KUKA KRL program: ps_l_res_c1.src, ps_l_res_c1.dat

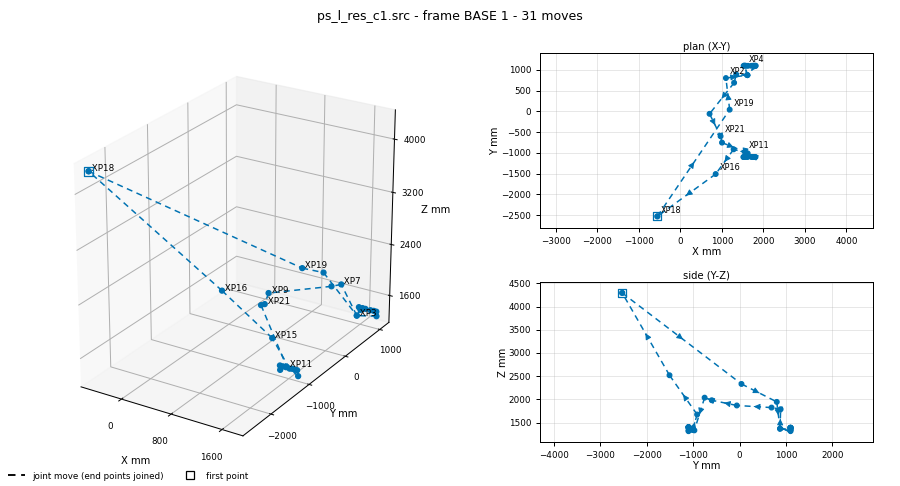
[picture p0: tool path of ps_l_res_c1.src in frame BASE 1, 31 of 31 moves have a stored position in this frame; points joined in program order, loops and branches not executed]
--- ps_l_res_c1.src ---
&ACCESS RVO1
&REL 7
&COMMENT SOLDA GUN C1 SEM GRIPPER
&PARAM DISKPATH = KRC:\R1\Program
DEF ps_l_res_c1( )
;FOLD INI
;FOLD SPOTTECH INI
USERSPOT(#INIT)
;ENDFOLD (SPOTTECH INI)
;FOLD GRIPPERTECH INI
USER_GRP(0,DUMMY,DUMMY,GDEFAULT)
;ENDFOLD (GRIPPERTECH INI)
  ;FOLD USER INI
    ;Make your modifications here

  ;ENDFOLD (USER INI)
;ENDFOLD (INI)

; Caracterização dos meios de produção:
; Versão Atual:
; 15/07/2013 12:00 Name: P13.050-R5 CHANGES: Solda Respot Actros
; C1 LTA/LTB/MGS/MGSB

chk_w1_wechs_ok ( )      ; CHECK FERRAMENTA: C1

;FOLD PTP P18 CONT Vel=100 % PDAT31 Tool[1]:Gun C1 Base[1]:ACTROS;%{PE}%R 8.2.20,%MKUKATPBASIS,%CMOVE,%VPTP,%P 1:PTP, 2:P18, 3:C_DIS, 5:100, 7:PDAT31
$BWDSTART=FALSE
PDAT_ACT=PPDAT31
FDAT_ACT=FP18
BAS(#PTP_PARAMS,100)
PTP XP18 C_DIS
;ENDFOLD

if MaxStandMenge (1) then
 MaxStandmengeErreicht (1)
endif

IF (NOT(GHOST())) THEN
if Elektrodenwechsel (1) then
 e_fraes1 ()
endif
ENDIF

;FOLD PTP P19 CONT Vel=100 % PDAT32 Tool[1]:Gun C1 Base[1]:ACTROS;%{PE}%R 8.2.20,%MKUKATPBASIS,%CMOVE,%VPTP,%P 1:PTP, 2:P19, 3:C_DIS, 5:100, 7:PDAT32
$BWDSTART=FALSE
PDAT_ACT=PPDAT32
FDAT_ACT=FP19
BAS(#PTP_PARAMS,100)
PTP XP19 C_DIS
;ENDFOLD

;FOLD OUT 3334 'R5 solicita lib soldar respot' State=TRUE ;%{PE}%R 8.2.20,%MKUKATPBASIS,%COUT,%VOUTX,%P 2:3334, 3:R5 solicita lib soldar respot, 5:TRUE, 6:
$OUT[3334]=TRUE
;ENDFOLD
;FOLD OUT 3337 'R5 retirando garra Geo' State=TRUE ;%{PE}%R 8.2.20,%MKUKATPBASIS,%COUT,%VOUTX,%P 2:3337, 3:R5 retirando garra Geo, 5:TRUE, 6:
$OUT[3337]=TRUE
;ENDFOLD
;FOLD WAIT FOR ( IN 3334 'Aguarda lib soldar respot' );%{PE}%R 8.2.20,%MKUKATPBASIS,%CEXT_WAIT_FOR,%VEXT_WAIT_FOR,%P 2:, 4:, 5:$IN, 6:3334, 7:Aguarda lib soldar respot, 9:
WAIT FOR  ( $IN[3334] )
;ENDFOLD
;FOLD OUT 3334 'R5 solicita lib soldar respot' State=FALSE ;%{PE}%R 8.2.20,%MKUKATPBASIS,%COUT,%VOUTX,%P 2:3334, 3:R5 solicita lib soldar respot, 5:FALSE, 6:
$OUT[3334]=FALSE
;ENDFOLD
;FOLD OUT 3337 'R5 retirando garra Geo' State=FALSE ;%{PE}%R 8.2.20,%MKUKATPBASIS,%COUT,%VOUTX,%P 2:3337, 3:R5 retirando garra Geo, 5:FALSE, 6:
$OUT[3337]=FALSE
;ENDFOLD
;FOLD OUT 3338 'R5 solda geometria concluida' State=FALSE ;%{PE}%R 8.2.20,%MKUKATPBASIS,%COUT,%VOUTX,%P 2:3338, 3:R5 solda geometria concluida, 5:FALSE, 6:
$OUT[3338]=FALSE
;ENDFOLD
;FOLD OUT 3348 'Fora area GEOBOX' State=FALSE ;%{PE}%R 8.2.20,%MKUKATPBASIS,%COUT,%VOUTX,%P 2:3348, 3:Fora area GEOBOX, 5:FALSE, 6:
$OUT[3348]=FALSE
;ENDFOLD
;FOLD  ;%{PE}%R 8.2.20,%MKUKATPBASIS,%CCOMMENT,%VNORMAL,%P 2:
;ENDFOLD
;FOLD PTP P2 CONT Vel=100 % PDAT2 Tool[1]:Gun C1 Base[1]:ACTROS;%{PE}%R 8.2.20,%MKUKATPBASIS,%CMOVE,%VPTP,%P 1:PTP, 2:P2, 3:C_DIS, 5:100, 7:PDAT2
$BWDSTART=FALSE
PDAT_ACT=PPDAT2
FDAT_ACT=FP2
BAS(#PTP_PARAMS,100)
PTP XP2 C_DIS
;ENDFOLD
;FOLD PTP P3 CONT Vel=100 % PDAT3 Tool[1]:Gun C1 Base[1]:ACTROS;%{PE}%R 8.2.20,%MKUKATPBASIS,%CMOVE,%VPTP,%P 1:PTP, 2:P3, 3:C_DIS, 5:100, 7:PDAT3
$BWDSTART=FALSE
PDAT_ACT=PPDAT3
FDAT_ACT=FP3
BAS(#PTP_PARAMS,100)
PTP XP3 C_DIS
;ENDFOLD
;FOLD PTP P4 CONT Vel=100 % PDAT4 Tool[1]:Gun C1 Base[1]:ACTROS;%{PE}%R 8.2.20,%MKUKATPBASIS,%CMOVE,%VPTP,%P 1:PTP, 2:P4, 3:C_DIS, 5:100, 7:PDAT4
$BWDSTART=FALSE
PDAT_ACT=PPDAT4
FDAT_ACT=FP4
BAS(#PTP_PARAMS,100)
PTP XP4 C_DIS
;ENDFOLD

;FOLD ; swp_60_5662;%{PE}%R 8.2.20,%MKUKATPBASIS,%CCOMMENT,%VNORMAL,%P 2:swp_60_5662
;ENDFOLD
;FOLD PTP Xswp_60_5662 PDAT5 SPOT Gun=1 RETR OPN PgNo1=38 ACTIVE=1 Tool[1]:Gun C1 Base[1]:ACTROS;%{PE}%R 8.2.2,%MKUKATPSPOT,%CSPOT,%VPTP,%P 1:PTP, 2:Xswp_60_5662, 3:, 5:100, 7:PDAT5, 10:1, 12:#FIRST, 14:#OPN, 16:38, 18:1, 20:0, 22:0, 24:1, 25:NORMAL
$BWDSTART=FALSE
PDAT_ACT=PPDAT5
FDAT_ACT=FXswp_60_5662
BAS(#PTP_PARAMS,PPDAT5.VEL)
S_ACT.GUN=1
S_ACT.PAIR=SDEFAULT.PAIR
S_ACT.RETR=#OPN
S_ACT.CLO_TM=1
S_ACT.PGNO1=38
S_ACT.PGNO2=SDEFAULT.PGNO2
S_ACT.PRESS1=SDEFAULT.PRESS1
S_ACT.PRESS2=SDEFAULT.PRESS2
S_READY=FALSE
PTP XXswp_60_5662
USERSPOT(#SPOT, S_ACT)
WAIT FOR S_READY
;ENDFOLD

;FOLD ; swp_60_5664;%{PE}%R 8.2.20,%MKUKATPBASIS,%CCOMMENT,%VNORMAL,%P 2:swp_60_5664
;ENDFOLD
;FOLD PTP Xswp_60_5664 PDAT7 SPOT Gun=1 RETR CLS PgNo1=39 ACTIVE=1 Tool[1]:Gun C1 Base[1]:ACTROS;%{PE}%R 8.2.2,%MKUKATPSPOT,%CSPOT,%VPTP,%P 1:PTP, 2:Xswp_60_5664, 3:, 5:100, 7:PDAT7, 10:1, 12:#FIRST, 14:#CLO, 16:39, 18:1, 20:0, 22:0, 24:1, 25:NORMAL
$BWDSTART=FALSE
PDAT_ACT=PPDAT7
FDAT_ACT=FXswp_60_5664
BAS(#PTP_PARAMS,PPDAT7.VEL)
S_ACT.GUN=1
S_ACT.PAIR=SDEFAULT.PAIR
S_ACT.RETR=#CLO
S_ACT.CLO_TM=1
S_ACT.PGNO1=39
S_ACT.PGNO2=SDEFAULT.PGNO2
S_ACT.PRESS1=SDEFAULT.PRESS1
S_ACT.PRESS2=SDEFAULT.PRESS2
S_READY=FALSE
PTP XXswp_60_5664
USERSPOT(#SPOT, S_ACT)
WAIT FOR S_READY
;ENDFOLD

;FOLD ; swp_60_5666;%{PE}%R 8.2.20,%MKUKATPBASIS,%CCOMMENT,%VNORMAL,%P 2:swp_60_5666
;ENDFOLD
;FOLD PTP Xswp_60_5666 PDAT6 SPOT Gun=1 RETR CLS PgNo1=40 ACTIVE=1 Tool[1]:Gun C1 Base[1]:ACTROS;%{PE}%R 8.2.2,%MKUKATPSPOT,%CSPOT,%VPTP,%P 1:PTP, 2:Xswp_60_5666, 3:, 5:100, 7:PDAT6, 10:1, 12:#FIRST, 14:#CLO, 16:40, 18:1, 20:0, 22:0, 24:1, 25:NORMAL
$BWDSTART=FALSE
PDAT_ACT=PPDAT6
FDAT_ACT=FXswp_60_5666
BAS(#PTP_PARAMS,PPDAT6.VEL)
S_ACT.GUN=1
S_ACT.PAIR=SDEFAULT.PAIR
S_ACT.RETR=#CLO
S_ACT.CLO_TM=1
S_ACT.PGNO1=40
S_ACT.PGNO2=SDEFAULT.PGNO2
S_ACT.PRESS1=SDEFAULT.PRESS1
S_ACT.PRESS2=SDEFAULT.PRESS2
S_READY=FALSE
PTP XXswp_60_5666
USERSPOT(#SPOT, S_ACT)
WAIT FOR S_READY
;ENDFOLD

;FOLD ; swp_60_5670;%{PE}%R 8.2.20,%MKUKATPBASIS,%CCOMMENT,%VNORMAL,%P 2:swp_60_5670
;ENDFOLD
;FOLD PTP Xswp_60_5670 PDAT8 SPOT Gun=1 RETR CLS PgNo1=41 ACTIVE=1 Tool[1]:Gun C1 Base[1]:ACTROS;%{PE}%R 8.2.2,%MKUKATPSPOT,%CSPOT,%VPTP,%P 1:PTP, 2:Xswp_60_5670, 3:, 5:100, 7:PDAT8, 10:1, 12:#FIRST, 14:#CLO, 16:41, 18:1, 20:0, 22:0, 24:1, 25:NORMAL
$BWDSTART=FALSE
PDAT_ACT=PPDAT8
FDAT_ACT=FXswp_60_5670
BAS(#PTP_PARAMS,PPDAT8.VEL)
S_ACT.GUN=1
S_ACT.PAIR=SDEFAULT.PAIR
S_ACT.RETR=#CLO
S_ACT.CLO_TM=1
S_ACT.PGNO1=41
S_ACT.PGNO2=SDEFAULT.PGNO2
S_ACT.PRESS1=SDEFAULT.PRESS1
S_ACT.PRESS2=SDEFAULT.PRESS2
S_READY=FALSE
PTP XXswp_60_5670
USERSPOT(#SPOT, S_ACT)
WAIT FOR S_READY
;ENDFOLD

;FOLD ; swp_60_5672;%{PE}%R 8.2.20,%MKUKATPBASIS,%CCOMMENT,%VNORMAL,%P 2:swp_60_5672
;ENDFOLD
;FOLD PTP SWP_60_5672 PDAT30 SPOT Gun=1 RETR CLS PgNo1=42 ACTIVE=1 Tool[1]:Gun C1 Base[1]:ACTROS;%{PE}%R 8.2.2,%MKUKATPSPOT,%CSPOT,%VPTP,%P 1:PTP, 2:SWP_60_5672, 3:, 5:100, 7:PDAT30, 10:1, 12:#FIRST, 14:#CLO, 16:42, 18:1, 20:0, 22:0, 24:1, 25:NORMAL
$BWDSTART=FALSE
PDAT_ACT=PPDAT30
FDAT_ACT=FSWP_60_5672
BAS(#PTP_PARAMS,PPDAT30.VEL)
S_ACT.GUN=1
S_ACT.PAIR=SDEFAULT.PAIR
S_ACT.RETR=#CLO
S_ACT.CLO_TM=1
S_ACT.PGNO1=42
S_ACT.PGNO2=SDEFAULT.PGNO2
S_ACT.PRESS1=SDEFAULT.PRESS1
S_ACT.PRESS2=SDEFAULT.PRESS2
S_READY=FALSE
PTP XSWP_60_5672
USERSPOT(#SPOT, S_ACT)
WAIT FOR S_READY
;ENDFOLD

;FOLD ; swp_60_5674;%{PE}%R 8.2.20,%MKUKATPBASIS,%CCOMMENT,%VNORMAL,%P 2:swp_60_5674
;ENDFOLD
;FOLD PTP Xswp_60_5674 PDAT10 SPOT Gun=1 RETR CLS PgNo1=43 ACTIVE=1 Tool[1]:Gun C1 Base[1]:ACTROS;%{PE}%R 8.2.2,%MKUKATPSPOT,%CSPOT,%VPTP,%P 1:PTP, 2:Xswp_60_5674, 3:, 5:100, 7:PDAT10, 10:1, 12:#FIRST, 14:#CLO, 16:43, 18:1, 20:0, 22:0, 24:1, 25:NORMAL
$BWDSTART=FALSE
PDAT_ACT=PPDAT10
FDAT_ACT=FXswp_60_5674
BAS(#PTP_PARAMS,PPDAT10.VEL)
S_ACT.GUN=1
S_ACT.PAIR=SDEFAULT.PAIR
S_ACT.RETR=#CLO
S_ACT.CLO_TM=1
S_ACT.PGNO1=43
S_ACT.PGNO2=SDEFAULT.PGNO2
S_ACT.PRESS1=SDEFAULT.PRESS1
S_ACT.PRESS2=SDEFAULT.PRESS2
S_READY=FALSE
PTP XXswp_60_5674
USERSPOT(#SPOT, S_ACT)
WAIT FOR S_READY
;ENDFOLD

;FOLD PTP P5 CONT Vel=100 % PDAT11 Tool[1]:Gun C1 Base[1]:ACTROS;%{PE}%R 8.2.20,%MKUKATPBASIS,%CMOVE,%VPTP,%P 1:PTP, 2:P5, 3:C_DIS, 5:100, 7:PDAT11
$BWDSTART=FALSE
PDAT_ACT=PPDAT11
FDAT_ACT=FP5
BAS(#PTP_PARAMS,100)
PTP XP5 C_DIS
;ENDFOLD
;FOLD PTP P6 CONT Vel=100 % PDAT12 Tool[1]:Gun C1 Base[1]:ACTROS;%{PE}%R 8.2.20,%MKUKATPBASIS,%CMOVE,%VPTP,%P 1:PTP, 2:P6, 3:C_DIS, 5:100, 7:PDAT12
$BWDSTART=FALSE
PDAT_ACT=PPDAT12
FDAT_ACT=FP6
BAS(#PTP_PARAMS,100)
PTP XP6 C_DIS
;ENDFOLD
;FOLD PTP P7 CONT Vel=100 % PDAT13 Tool[1]:Gun C1 Base[1]:ACTROS;%{PE}%R 8.2.20,%MKUKATPBASIS,%CMOVE,%VPTP,%P 1:PTP, 2:P7, 3:C_DIS, 5:100, 7:PDAT13
$BWDSTART=FALSE
PDAT_ACT=PPDAT13
FDAT_ACT=FP7
BAS(#PTP_PARAMS,100)
PTP XP7 C_DIS
;ENDFOLD
;FOLD PTP P22 CONT Vel=100 % PDAT35 Tool[1]:Gun C1 Base[1]:ACTROS;%{PE}%R 8.2.20,%MKUKATPBASIS,%CMOVE,%VPTP,%P 1:PTP, 2:P22, 3:C_DIS, 5:100, 7:PDAT35
$BWDSTART=FALSE
PDAT_ACT=PPDAT35
FDAT_ACT=FP22
BAS(#PTP_PARAMS,100)
PTP XP22 C_DIS
;ENDFOLD
;FOLD PTP P9 CONT Vel=100 % PDAT15 Tool[1]:Gun C1 Base[1]:ACTROS;%{PE}%R 8.2.20,%MKUKATPBASIS,%CMOVE,%VPTP,%P 1:PTP, 2:P9, 3:C_DIS, 5:100, 7:PDAT15
$BWDSTART=FALSE
PDAT_ACT=PPDAT15
FDAT_ACT=FP9
BAS(#PTP_PARAMS,100)
PTP XP9 C_DIS
;ENDFOLD
;FOLD PTP P21 CONT Vel=100 % PDAT34 Tool[1]:Gun C1 Base[1]:ACTROS;%{PE}%R 8.2.20,%MKUKATPBASIS,%CMOVE,%VPTP,%P 1:PTP, 2:P21, 3:C_DIS, 5:100, 7:PDAT34
$BWDSTART=FALSE
PDAT_ACT=PPDAT34
FDAT_ACT=FP21
BAS(#PTP_PARAMS,100)
PTP XP21 C_DIS
;ENDFOLD
;FOLD PTP P10 CONT Vel=100 % PDAT16 Tool[1]:Gun C1 Base[1]:ACTROS;%{PE}%R 8.2.20,%MKUKATPBASIS,%CMOVE,%VPTP,%P 1:PTP, 2:P10, 3:C_DIS, 5:100, 7:PDAT16
$BWDSTART=FALSE
PDAT_ACT=PPDAT16
FDAT_ACT=FP10
BAS(#PTP_PARAMS,100)
PTP XP10 C_DIS
;ENDFOLD
;FOLD PTP P11 CONT Vel=100 % PDAT17 Tool[1]:Gun C1 Base[1]:ACTROS;%{PE}%R 8.2.20,%MKUKATPBASIS,%CMOVE,%VPTP,%P 1:PTP, 2:P11, 3:C_DIS, 5:100, 7:PDAT17
$BWDSTART=FALSE
PDAT_ACT=PPDAT17
FDAT_ACT=FP11
BAS(#PTP_PARAMS,100)
PTP XP11 C_DIS
;ENDFOLD
;FOLD PTP P12 CONT Vel=100 % PDAT18 Tool[1]:Gun C1 Base[1]:ACTROS;%{PE}%R 8.2.20,%MKUKATPBASIS,%CMOVE,%VPTP,%P 1:PTP, 2:P12, 3:C_DIS, 5:100, 7:PDAT18
$BWDSTART=FALSE
PDAT_ACT=PPDAT18
FDAT_ACT=FP12
BAS(#PTP_PARAMS,100)
PTP XP12 C_DIS
;ENDFOLD

;FOLD ; swp_60_5661;%{PE}%R 8.2.20,%MKUKATPBASIS,%CCOMMENT,%VNORMAL,%P 2:swp_60_5661
;ENDFOLD
;FOLD PTP Xswp_60_5661 PDAT19 SPOT Gun=1 RETR CLS PgNo1=44 ACTIVE=1 Tool[1]:Gun C1 Base[1]:ACTROS;%{PE}%R 8.2.2,%MKUKATPSPOT,%CSPOT,%VPTP,%P 1:PTP, 2:Xswp_60_5661, 3:, 5:100, 7:PDAT19, 10:1, 12:#FIRST, 14:#CLO, 16:44, 18:1, 20:0, 22:0, 24:1, 25:NORMAL
$BWDSTART=FALSE
PDAT_ACT=PPDAT19
FDAT_ACT=FXswp_60_5661
BAS(#PTP_PARAMS,PPDAT19.VEL)
S_ACT.GUN=1
S_ACT.PAIR=SDEFAULT.PAIR
S_ACT.RETR=#CLO
S_ACT.CLO_TM=1
S_ACT.PGNO1=44
S_ACT.PGNO2=SDEFAULT.PGNO2
S_ACT.PRESS1=SDEFAULT.PRESS1
S_ACT.PRESS2=SDEFAULT.PRESS2
S_READY=FALSE
PTP XXswp_60_5661
USERSPOT(#SPOT, S_ACT)
WAIT FOR S_READY
;ENDFOLD

;FOLD ; swp_60_5663;%{PE}%R 8.2.20,%MKUKATPBASIS,%CCOMMENT,%VNORMAL,%P 2:swp_60_5663
;ENDFOLD
;FOLD PTP Xswp_60_5663 PDAT20 SPOT Gun=1 RETR CLS PgNo1=45 ACTIVE=1 Tool[1]:Gun C1 Base[1]:ACTROS;%{PE}%R 8.2.2,%MKUKATPSPOT,%CSPOT,%VPTP,%P 1:PTP, 2:Xswp_60_5663, 3:, 5:100, 7:PDAT20, 10:1, 12:#FIRST, 14:#CLO, 16:45, 18:1, 20:0, 22:0, 24:1, 25:NORMAL
$BWDSTART=FALSE
PDAT_ACT=PPDAT20
FDAT_ACT=FXswp_60_5663
BAS(#PTP_PARAMS,PPDAT20.VEL)
S_ACT.GUN=1
S_ACT.PAIR=SDEFAULT.PAIR
S_ACT.RETR=#CLO
S_ACT.CLO_TM=1
S_ACT.PGNO1=45
S_ACT.PGNO2=SDEFAULT.PGNO2
S_ACT.PRESS1=SDEFAULT.PRESS1
S_ACT.PRESS2=SDEFAULT.PRESS2
S_READY=FALSE
PTP XXswp_60_5663
USERSPOT(#SPOT, S_ACT)
WAIT FOR S_READY
;ENDFOLD

;FOLD ; swp_60_5665;%{PE}%R 8.2.20,%MKUKATPBASIS,%CCOMMENT,%VNORMAL,%P 2:swp_60_5665
;ENDFOLD
;FOLD PTP Xswp_60_5665 PDAT21 SPOT Gun=1 RETR CLS PgNo1=46 ACTIVE=1 Tool[1]:Gun C1 Base[1]:ACTROS;%{PE}%R 8.2.2,%MKUKATPSPOT,%CSPOT,%VPTP,%P 1:PTP, 2:Xswp_60_5665, 3:, 5:100, 7:PDAT21, 10:1, 12:#FIRST, 14:#CLO, 16:46, 18:1, 20:0, 22:0, 24:1, 25:NORMAL
$BWDSTART=FALSE
PDAT_ACT=PPDAT21
FDAT_ACT=FXswp_60_5665
BAS(#PTP_PARAMS,PPDAT21.VEL)
S_ACT.GUN=1
S_ACT.PAIR=SDEFAULT.PAIR
S_ACT.RETR=#CLO
S_ACT.CLO_TM=1
S_ACT.PGNO1=46
S_ACT.PGNO2=SDEFAULT.PGNO2
S_ACT.PRESS1=SDEFAULT.PRESS1
S_ACT.PRESS2=SDEFAULT.PRESS2
S_READY=FALSE
PTP XXswp_60_5665
USERSPOT(#SPOT, S_ACT)
WAIT FOR S_READY
;ENDFOLD

;FOLD ; swp_60_5669;%{PE}%R 8.2.20,%MKUKATPBASIS,%CCOMMENT,%VNORMAL,%P 2:swp_60_5669
;ENDFOLD
;FOLD PTP Xswp_60_5669 PDAT22 SPOT Gun=1 RETR CLS PgNo1=47 ACTIVE=1 Tool[1]:Gun C1 Base[1]:ACTROS;%{PE}%R 8.2.2,%MKUKATPSPOT,%CSPOT,%VPTP,%P 1:PTP, 2:Xswp_60_5669, 3:, 5:100, 7:PDAT22, 10:1, 12:#FIRST, 14:#CLO, 16:47, 18:1, 20:0, 22:0, 24:1, 25:NORMAL
$BWDSTART=FALSE
PDAT_ACT=PPDAT22
FDAT_ACT=FXswp_60_5669
BAS(#PTP_PARAMS,PPDAT22.VEL)
S_ACT.GUN=1
S_ACT.PAIR=SDEFAULT.PAIR
S_ACT.RETR=#CLO
S_ACT.CLO_TM=1
S_ACT.PGNO1=47
S_ACT.PGNO2=SDEFAULT.PGNO2
S_ACT.PRESS1=SDEFAULT.PRESS1
S_ACT.PRESS2=SDEFAULT.PRESS2
S_READY=FALSE
PTP XXswp_60_5669
USERSPOT(#SPOT, S_ACT)
WAIT FOR S_READY
;ENDFOLD

;FOLD ; swp_60_5671;%{PE}%R 8.2.20,%MKUKATPBASIS,%CCOMMENT,%VNORMAL,%P 2:swp_60_5671
;ENDFOLD
;FOLD PTP Xswp_60_5671 PDAT23 SPOT Gun=1 RETR CLS PgNo1=48 ACTIVE=1 Tool[1]:Gun C1 Base[1]:ACTROS;%{PE}%R 8.2.2,%MKUKATPSPOT,%CSPOT,%VPTP,%P 1:PTP, 2:Xswp_60_5671, 3:, 5:100, 7:PDAT23, 10:1, 12:#FIRST, 14:#CLO, 16:48, 18:1, 20:0, 22:0, 24:1, 25:NORMAL
$BWDSTART=FALSE
PDAT_ACT=PPDAT23
FDAT_ACT=FXswp_60_5671
BAS(#PTP_PARAMS,PPDAT23.VEL)
S_ACT.GUN=1
S_ACT.PAIR=SDEFAULT.PAIR
S_ACT.RETR=#CLO
S_ACT.CLO_TM=1
S_ACT.PGNO1=48
S_ACT.PGNO2=SDEFAULT.PGNO2
S_ACT.PRESS1=SDEFAULT.PRESS1
S_ACT.PRESS2=SDEFAULT.PRESS2
S_READY=FALSE
PTP XXswp_60_5671
USERSPOT(#SPOT, S_ACT)
WAIT FOR S_READY
;ENDFOLD

;FOLD ; swp_60_5673;%{PE}%R 8.2.20,%MKUKATPBASIS,%CCOMMENT,%VNORMAL,%P 2:swp_60_5673
;ENDFOLD
;FOLD PTP Xswp_60_5673 PDAT24 SPOT Gun=1 RETR OPN PgNo1=49 ACTIVE=1 Tool[1]:Gun C1 Base[1]:ACTROS;%{PE}%R 8.2.2,%MKUKATPSPOT,%CSPOT,%VPTP,%P 1:PTP, 2:Xswp_60_5673, 3:, 5:100, 7:PDAT24, 10:1, 12:#FIRST, 14:#OPN, 16:49, 18:1, 20:0, 22:0, 24:1, 25:NORMAL
$BWDSTART=FALSE
PDAT_ACT=PPDAT24
FDAT_ACT=FXswp_60_5673
BAS(#PTP_PARAMS,PPDAT24.VEL)
S_ACT.GUN=1
S_ACT.PAIR=SDEFAULT.PAIR
S_ACT.RETR=#OPN
S_ACT.CLO_TM=1
S_ACT.PGNO1=49
S_ACT.PGNO2=SDEFAULT.PGNO2
S_ACT.PRESS1=SDEFAULT.PRESS1
S_ACT.PRESS2=SDEFAULT.PRESS2
S_READY=FALSE
PTP XXswp_60_5673
USERSPOT(#SPOT, S_ACT)
WAIT FOR S_READY
;ENDFOLD

;FOLD PTP P13 CONT Vel=100 % PDAT25 Tool[1]:Gun C1 Base[1]:ACTROS;%{PE}%R 8.2.20,%MKUKATPBASIS,%CMOVE,%VPTP,%P 1:PTP, 2:P13, 3:C_DIS, 5:100, 7:PDAT25
$BWDSTART=FALSE
PDAT_ACT=PPDAT25
FDAT_ACT=FP13
BAS(#PTP_PARAMS,100)
PTP XP13 C_DIS
;ENDFOLD
;FOLD PTP P14 CONT Vel=100 % PDAT26 Tool[1]:Gun C1 Base[1]:ACTROS;%{PE}%R 8.2.20,%MKUKATPBASIS,%CMOVE,%VPTP,%P 1:PTP, 2:P14, 3:C_DIS, 5:100, 7:PDAT26
$BWDSTART=FALSE
PDAT_ACT=PPDAT26
FDAT_ACT=FP14
BAS(#PTP_PARAMS,100)
PTP XP14 C_DIS
;ENDFOLD
;FOLD PTP P15 CONT Vel=100 % PDAT27 Tool[1]:Gun C1 Base[1]:ACTROS;%{PE}%R 8.2.20,%MKUKATPBASIS,%CMOVE,%VPTP,%P 1:PTP, 2:P15, 3:C_DIS, 5:100, 7:PDAT27
$BWDSTART=FALSE
PDAT_ACT=PPDAT27
FDAT_ACT=FP15
BAS(#PTP_PARAMS,100)
PTP XP15 C_DIS
;ENDFOLD
;FOLD PTP P16 CONT Vel=100 % PDAT28 Tool[1]:Gun C1 Base[1]:ACTROS;%{PE}%R 8.2.20,%MKUKATPBASIS,%CMOVE,%VPTP,%P 1:PTP, 2:P16, 3:C_DIS, 5:100, 7:PDAT28
$BWDSTART=FALSE
PDAT_ACT=PPDAT28
FDAT_ACT=FP16
BAS(#PTP_PARAMS,100)
PTP XP16 C_DIS
;ENDFOLD
;FOLD  ;%{PE}%R 8.2.20,%MKUKATPBASIS,%CCOMMENT,%VNORMAL,%P 2:
;ENDFOLD
IF (NOT(GHOST())) THEN
if FraesAnf (1) then
f_fraes1 ()
endif
ENDIF

;FOLD OUT 3348 'Fora area GEOBOX' State=TRUE ;%{PE}%R 8.2.20,%MKUKATPBASIS,%COUT,%VOUTX,%P 2:3348, 3:Fora area GEOBOX, 5:TRUE, 6:
$OUT[3348]=TRUE
;ENDFOLD

;FOLD PTP P0 CONT Vel=100 % PDAT0 Tool[1]:Gun C1 Base[1]:ACTROS;%{PE}%R 8.2.20,%MKUKATPBASIS,%CMOVE,%VPTP,%P 1:PTP, 2:P0, 3:C_DIS, 5:100, 7:PDAT0
$BWDSTART=FALSE
PDAT_ACT=PPDAT0
FDAT_ACT=FP0
BAS(#PTP_PARAMS,100)
PTP XP0 C_DIS
;ENDFOLD

END

--- ps_l_res_c1.dat ---
&ACCESS RVO1
&REL 7
&COMMENT SOLDA GUN C1 SEM GRIPPER
&PARAM DISKPATH = KRC:\R1\Program
DEFDAT  ps_l_res_c1
;FOLD EXTERNAL DECLARATIONS;%{PE}%MKUKATPBASIS,%CEXT,%VCOMMON,%P
;FOLD GRIPPERTECH EXT
EXT  H50 (INT  :IN,INT  :IN,INT  :IN,GRP_TYP  :IN )
;ENDFOLD (GRIPPERTECH EXT)
;FOLD SPOTTECH EXT
EXT  USERSPOT (S_COMMAND  :IN,SPOT_TYPE  :IN )
;ENDFOLD (SPOTTECH EXT)
;FOLD BASISTECH EXT;%{PE}%MKUKATPBASIS,%CEXT,%VEXT,%P
EXT  BAS (BAS_COMMAND  :IN,REAL  :IN )
DECL INT SUCCESS
;ENDFOLD (BASISTECH EXT)
;FOLD USER EXT;%{E}%MKUKATPUSER,%CEXT,%VEXT,%P
;Make your modifications here

;ENDFOLD (USER EXT)
;ENDFOLD (EXTERNAL DECLARATIONS)

;# ============ START PATH : swp_p13050r5_l_res_c1 =============
DECL FDAT Fswp_60_5672={TOOL_NO 1,BASE_NO 1,IPO_FRAME #BASE,POINT2[] " "}
DECL E6POS Xswp_60_5672={X 1762.00098,Y 1101.5,Z 1386.453,A 0.0,B -90.0000534,C 89.9999619,S 2,T 40,E1 0.0,E2 0.0,E3 0.0,E4 0.0,E5 0.0,E6 0.0}
DECL BASIS_SUGG_T LAST_BASIS={POINT1[] "P22                     ",POINT2[] "P22                     ",CP_PARAMS[] "CPDAT0                  ",PTP_PARAMS[] "PDAT35                  ",CONT[] "C_DIS                   ",CP_VEL[] "2.0                     ",PTP_VEL[] "100                     ",SYNC_PARAMS[] "SYNCDAT                 ",SPL_NAME[] "S0                      "}
DECL E6POS XP2={X 1095.00696,Y 801.749573,Z 1944.729,A 111.118202,B -70.3253708,C -17.7125702,S 2,T 10,E1 0.0,E2 0.0,E3 0.0,E4 0.0,E5 0.0,E6 0.0}
DECL FDAT FP2={TOOL_NO 1,BASE_NO 1,IPO_FRAME #BASE,POINT2[] " ",TQ_STATE FALSE}
DECL PDAT PPDAT2={VEL 100.0,ACC 100.0,APO_DIST 100.0,APO_MODE #CDIS}
DECL E6POS XP3={X 1613.15405,Y 872.018494,Z 1367.10706,A 93.5968628,B -78.2830963,C -15.5704298,S 2,T 8,E1 0.0,E2 0.0,E3 0.0,E4 0.0,E5 0.0,E6 0.0}
DECL FDAT FP3={TOOL_NO 1,BASE_NO 1,IPO_FRAME #BASE,POINT2[] " ",TQ_STATE FALSE}
DECL PDAT PPDAT3={VEL 100.0,ACC 100.0,APO_DIST 100.0,APO_MODE #CDIS}
DECL E6POS XP4={X 1544.70605,Y 1103.80603,Z 1345.94702,A 178.820007,B -67.8129578,C -88.9299316,S 2,T 8,E1 0.0,E2 0.0,E3 0.0,E4 0.0,E5 0.0,E6 0.0}
DECL FDAT FP4={TOOL_NO 1,BASE_NO 1,IPO_FRAME #BASE,POINT2[] " ",TQ_STATE FALSE}
DECL PDAT PPDAT4={VEL 100.0,ACC 100.0,APO_DIST 100.0,APO_MODE #CDIS}
DECL SPOT_SUGG_T LAST_SPOT={GUN[] "1                       ",RETR_CMD[] "#CLO                    ",CHOISE[] "#FIRST                  ",CLO_TM[] "1                       ",PGNO1[] "1                       ",PRESS1[] "0                       ",PGNO2[] "1                       ",PRESS2[] "0                       ",SPOT_PARAMS[] "NORMAL                  "}
DECL E6POS XP5={X 1811.00305,Y 1098.526,Z 1314.68396,A -2.83520198,B -77.3528519,C 89.8615189,S 2,T 40,E1 0.0,E2 0.0,E3 0.0,E4 0.0,E5 0.0,E6 0.0}
DECL FDAT FP5={TOOL_NO 1,BASE_NO 1,IPO_FRAME #BASE,POINT2[] " ",TQ_STATE FALSE}
DECL PDAT PPDAT5={VEL 100.0,ACC 100.0,APO_DIST 100.0}
DECL E6POS XXSWP_60_5662={X 1522.03003,Y 1096.51196,Z 1386.07397,A 178.820007,B -67.8129807,C -88.9298935,S 2,T 8,E1 0.0,E2 0.0,E3 0.0,E4 0.0,E5 0.0,E6 0.0}
DECL FDAT FXswp_60_5662={TOOL_NO 1,BASE_NO 1,IPO_FRAME #BASE,POINT2[] " ",TQ_STATE FALSE}
DECL E6POS XXSWP_60_5666={X 1628.34094,Y 1097.005,Z 1386.10901,A 177.280197,B -87.5259018,C -87.3151703,S 2,T 8,E1 0.0,E2 0.0,E3 0.0,E4 0.0,E5 0.0,E6 0.0}
DECL FDAT FXswp_60_5666={TOOL_NO 1,BASE_NO 1,IPO_FRAME #BASE,POINT2[] " ",TQ_STATE FALSE}
DECL PDAT PPDAT6={VEL 100.0,ACC 100.0,APO_DIST 100.0}
DECL E6POS XXSWP_60_5664={X 1580.34399,Y 1096.995,Z 1386.07397,A 179.588806,B -73.3652573,C -89.6388931,S 2,T 8,E1 0.0,E2 0.0,E3 0.0,E4 0.0,E5 0.0,E6 0.0}
DECL FDAT FXswp_60_5664={TOOL_NO 1,BASE_NO 1,IPO_FRAME #BASE,POINT2[] " ",TQ_STATE FALSE}
DECL PDAT PPDAT7={VEL 100.0,ACC 100.0,APO_DIST 100.0}
DECL E6POS XXSWP_60_5670={X 1711.65002,Y 1096.99805,Z 1385.47205,A -0.72773689,B -89.7948227,C 90.5279617,S 2,T 40,E1 0.0,E2 0.0,E3 0.0,E4 0.0,E5 0.0,E6 0.0}
DECL FDAT FXswp_60_5670={TOOL_NO 1,BASE_NO 1,IPO_FRAME #BASE,POINT2[] " ",TQ_STATE FALSE}
DECL PDAT PPDAT8={VEL 100.0,ACC 100.0,APO_DIST 100.0}
DECL E6POS XXSWP_60_5674={X 1806.48206,Y 1098.36694,Z 1386.63904,A 0.302990288,B -85.8768768,C 89.5522385,S 2,T 40,E1 0.0,E2 0.0,E3 0.0,E4 0.0,E5 0.0,E6 0.0}
DECL FDAT FXswp_60_5674={TOOL_NO 1,BASE_NO 1,IPO_FRAME #BASE,POINT2[] " ",TQ_STATE FALSE}
DECL PDAT PPDAT10={VEL 100.0,ACC 100.0,APO_DIST 100.0}
DECL PDAT PPDAT11={VEL 100.0,ACC 100.0,APO_DIST 0.0,APO_MODE #CDIS}
DECL E6POS XP6={X 1613.15405,Y 872.018372,Z 1367.10706,A 93.5968781,B -78.2830963,C -15.5704498,S 2,T 8,E1 0.0,E2 0.0,E3 0.0,E4 0.0,E5 0.0,E6 0.0}
DECL FDAT FP6={TOOL_NO 1,BASE_NO 1,IPO_FRAME #BASE,POINT2[] " ",TQ_STATE FALSE}
DECL PDAT PPDAT12={VEL 100.0,ACC 100.0,APO_DIST 100.0,APO_MODE #CDIS}
DECL E6POS XP7={X 1342.65002,Y 884.754822,Z 1786.34302,A 96.2288818,B -69.3940735,C -12.7518902,S 2,T 10,E1 0.0,E2 0.0,E3 0.0,E4 0.0,E5 0.0,E6 0.0}
DECL FDAT FP7={TOOL_NO 1,BASE_NO 1,IPO_FRAME #BASE,POINT2[] " ",TQ_STATE FALSE}
DECL PDAT PPDAT13={VEL 100.0,ACC 100.0,APO_DIST 100.0,APO_MODE #CDIS}
DECL E6POS XP9={X 701.170227,Y -60.0373497,Z 1867.28796,A 177.365799,B -38.748539,C 3.98628807,S 2,T 2,E1 0.0,E2 0.0,E3 0.0,E4 0.0,E5 0.0,E6 0.0}
DECL FDAT FP9={TOOL_NO 1,BASE_NO 1,IPO_FRAME #BASE,POINT2[] " ",TQ_STATE FALSE}
DECL PDAT PPDAT15={VEL 100.0,ACC 100.0,APO_DIST 100.0,APO_MODE #CDIS}
DECL E6POS XP10={X 1001.27802,Y -754.350708,Z 2035.755,A -141.764297,B -62.2648811,C 46.2266808,S 2,T 35,E1 0.0,E2 0.0,E3 0.0,E4 0.0,E5 0.0,E6 0.0}
DECL FDAT FP10={TOOL_NO 1,BASE_NO 1,IPO_FRAME #BASE,POINT2[] " ",TQ_STATE FALSE}
DECL PDAT PPDAT16={VEL 100.0,ACC 100.0,APO_DIST 100.0,APO_MODE #CDIS}
DECL E6POS XP11={X 1551.125,Y -974.612,Z 1330.552,A 179.999496,B -69.9997787,C 90.000679,S 2,T 1,E1 0.0,E2 0.0,E3 0.0,E4 0.0,E5 0.0,E6 0.0}
DECL FDAT FP11={TOOL_NO 1,BASE_NO 1,IPO_FRAME #BASE,POINT2[] " ",TQ_STATE FALSE}
DECL PDAT PPDAT17={VEL 100.0,ACC 100.0,APO_DIST 100.0,APO_MODE #CDIS}
DECL E6POS XP12={X 1522.94299,Y -1101.51196,Z 1330.97205,A -179.999802,B -63.8368683,C 89.9998779,S 2,T 33,E1 0.0,E2 0.0,E3 0.0,E4 0.0,E5 0.0,E6 0.0}
DECL FDAT FP12={TOOL_NO 1,BASE_NO 1,IPO_FRAME #BASE,POINT2[] " ",TQ_STATE FALSE}
DECL PDAT PPDAT18={VEL 100.0,ACC 100.0,APO_DIST 100.0,APO_MODE #CDIS}
DECL E6POS XXSWP_60_5661={X 1517.96497,Y -1100.89404,Z 1396.78796,A -179.979599,B -68.3391418,C 90.0388794,S 2,T 1,E1 0.0,E2 0.0,E3 0.0,E4 0.0,E5 0.0,E6 0.0}
DECL FDAT FXswp_60_5661={TOOL_NO 1,BASE_NO 1,IPO_FRAME #BASE,POINT2[] " ",TQ_STATE FALSE}
DECL PDAT PPDAT19={VEL 100.0,ACC 100.0,APO_DIST 100.0}
DECL E6POS XXSWP_60_5663={X 1565.52698,Y -1100.92297,Z 1396.14099,A 179.975494,B -73.3556137,C 89.9738388,S 2,T 1,E1 0.0,E2 0.0,E3 0.0,E4 0.0,E5 0.0,E6 0.0}
DECL FDAT FXswp_60_5663={TOOL_NO 1,BASE_NO 1,IPO_FRAME #BASE,POINT2[] " ",TQ_STATE FALSE}
DECL PDAT PPDAT20={VEL 100.0,ACC 100.0,APO_DIST 100.0}
DECL E6POS XXSWP_60_5665={X 1614.38794,Y -1100.98999,Z 1396.22705,A -179.984497,B -82.937088,C 89.9861984,S 2,T 1,E1 0.0,E2 0.0,E3 0.0,E4 0.0,E5 0.0,E6 0.0}
DECL FDAT FXswp_60_5665={TOOL_NO 1,BASE_NO 1,IPO_FRAME #BASE,POINT2[] " ",TQ_STATE FALSE}
DECL PDAT PPDAT21={VEL 100.0,ACC 100.0,APO_DIST 100.0}
DECL E6POS XXSWP_60_5669={X 1712.51099,Y -1100.95801,Z 1399.25696,A -0.0001528258,B -43.399601,C -89.990799,S 2,T 1,E1 0.0,E2 0.0,E3 0.0,E4 0.0,E5 0.0,E6 0.0}
DECL FDAT FXswp_60_5669={TOOL_NO 1,BASE_NO 1,IPO_FRAME #BASE,POINT2[] " ",TQ_STATE FALSE}
DECL PDAT PPDAT22={VEL 100.0,ACC 100.0,APO_DIST 100.0}
DECL E6POS XXSWP_60_5671={X 1753.97595,Y -1100.96301,Z 1398.60706,A -0.000141054799,B -43.3987312,C -89.9908371,S 2,T 1,E1 0.0,E2 0.0,E3 0.0,E4 0.0,E5 0.0,E6 0.0}
DECL FDAT FXswp_60_5671={TOOL_NO 1,BASE_NO 1,IPO_FRAME #BASE,POINT2[] " ",TQ_STATE FALSE}
DECL PDAT PPDAT23={VEL 100.0,ACC 100.0,APO_DIST 100.0}
DECL E6POS XXSWP_60_5673={X 1790.78406,Y -1101.04102,Z 1398.62,A 0.106619902,B -45.0337105,C -89.9933167,S 2,T 1,E1 0.0,E2 0.0,E3 0.0,E4 0.0,E5 0.0,E6 0.0}
DECL FDAT FXswp_60_5673={TOOL_NO 1,BASE_NO 1,IPO_FRAME #BASE,POINT2[] " ",TQ_STATE FALSE}
DECL PDAT PPDAT24={VEL 100.0,ACC 100.0,APO_DIST 100.0}
DECL E6POS XP13={X 1807.65601,Y -1101.05396,Z 1312.65796,A 0.106279403,B -45.033699,C -89.9933624,S 2,T 1,E1 0.0,E2 0.0,E3 0.0,E4 0.0,E5 0.0,E6 0.0}
DECL FDAT FP13={TOOL_NO 1,BASE_NO 1,IPO_FRAME #BASE,POINT2[] " ",TQ_STATE FALSE}
DECL PDAT PPDAT25={VEL 100.0,ACC 100.0,APO_DIST 0.0,APO_MODE #CDIS}
DECL E6POS XP14={X 1619.82397,Y -1012.995,Z 1337.65002,A -88.065712,B -84.0612488,C 3.50928211,S 2,T 1,E1 0.0,E2 0.0,E3 0.0,E4 0.0,E5 0.0,E6 0.0}
DECL FDAT FP14={TOOL_NO 1,BASE_NO 1,IPO_FRAME #BASE,POINT2[] " ",TQ_STATE FALSE}
DECL PDAT PPDAT26={VEL 100.0,ACC 100.0,APO_DIST 100.0,APO_MODE #CDIS}
DECL E6POS XP15={X 1281.40405,Y -915.495789,Z 1672.53601,A -47.3513794,B -52.3629417,C -36.2565308,S 2,T 3,E1 0.0,E2 0.0,E3 0.0,E4 0.0,E5 0.0,E6 0.0}
DECL FDAT FP15={TOOL_NO 1,BASE_NO 1,IPO_FRAME #BASE,POINT2[] " ",TQ_STATE FALSE}
DECL PDAT PPDAT27={VEL 100.0,ACC 100.0,APO_DIST 100.0,APO_MODE #CDIS}
DECL E6POS XP16={X 848.661316,Y -1511.198,Z 2518.677,A -41.1533508,B -17.6754208,C -33.2526512,S 2,T 2,E1 0.0,E2 0.0,E3 0.0,E4 0.0,E5 0.0,E6 0.0}
DECL FDAT FP16={TOOL_NO 1,BASE_NO 1,IPO_FRAME #BASE,POINT2[] " ",TQ_STATE FALSE}
DECL PDAT PPDAT28={VEL 100.0,ACC 100.0,APO_DIST 100.0,APO_MODE #CDIS}
DECL PDAT PPDAT30={VEL 100.0,ACC 100.0,APO_DIST 100.0}
DECL E6POS XP18={X -556.388,Y -2530.85303,Z 4293.4668,A -119.594704,B -72.7613373,C 35.2795486,S 2,T 10,E1 0.0,E2 0.0,E3 0.0,E4 0.0,E5 0.0,E6 0.0}
DECL FDAT FP18={TOOL_NO 1,BASE_NO 1,IPO_FRAME #BASE,POINT2[] " ",TQ_STATE FALSE}
DECL PDAT PPDAT31={VEL 100.0,ACC 100.0,APO_DIST 100.0,APO_MODE #CDIS}
DECL E6POS XP19={X 1185.44604,Y 40.3466797,Z 2331.125,A 102.087601,B -50.1155281,C -25.5069199,S 2,T 10,E1 0.0,E2 0.0,E3 0.0,E4 0.0,E5 0.0,E6 0.0}
DECL FDAT FP19={TOOL_NO 1,BASE_NO 1,IPO_FRAME #BASE,POINT2[] " ",TQ_STATE FALSE}
DECL PDAT PPDAT32={VEL 100.0,ACC 100.0,APO_DIST 100.0,APO_MODE #CDIS}
DECL PDAT PPDAT0={VEL 100.0,ACC 100.0,APO_DIST 100.0,APO_MODE #CDIS}
DECL E6POS XP0={X -556.388,Y -2530.85303,Z 4293.4668,A -119.594704,B -72.7613373,C 35.2795486,S 2,T 10,E1 0.0,E2 0.0,E3 0.0,E4 0.0,E5 0.0,E6 0.0}
DECL FDAT FP0={TOOL_NO 1,BASE_NO 1,IPO_FRAME #BASE,POINT2[] " ",TQ_STATE FALSE}
DECL E6POS XP21={X 966.734375,Y -599.818176,Z 1980.02905,A -120.728302,B -57.2565994,C 6.44424295,S 2,T 3,E1 0.0,E2 0.0,E3 0.0,E4 0.0,E5 0.0,E6 0.0}
DECL FDAT FP21={TOOL_NO 1,BASE_NO 1,IPO_FRAME #BASE,POINT2[] " ",TQ_STATE FALSE}
DECL PDAT PPDAT34={VEL 100.0,ACC 100.0,APO_DIST 100.0,APO_MODE #CDIS}
DECL E6POS XP22={X 1292.90796,Y 688.473999,Z 1821.93298,A 87.622612,B -46.9129486,C 3.00523901,S 2,T 42,E1 0.0,E2 0.0,E3 0.0,E4 0.0,E5 0.0,E6 0.0}
DECL FDAT FP22={TOOL_NO 1,BASE_NO 1,IPO_FRAME #BASE,POINT2[] " ",TQ_STATE FALSE}
DECL PDAT PPDAT35={VEL 100.0,ACC 100.0,APO_DIST 100.0,APO_MODE #CDIS}
ENDDAT
